// TIA Portal V18 export
TYPE "Rework_ShW"
// stored: IsFailsafeCompliant false
   STRUCT
      Trigger : Bool;
      Result : Int;
      Completed : Bool;
   END_STRUCT;
END_TYPE
